// TIA Portal V19 export
DATA_BLOCK "AI SCALING DB"   // DB5
{ S7_Optimized_Access := 'TRUE' }
// stored: MemoryReserve 100
   VAR RETAIN
      MIN : Struct
         "SYRUP VESSEL TEMP SENSOR" : Real := -50.0;
         "PREMIXING VESSEL TEMP SENSOR" : Real := -50.0;
         "SUGAR VESSEL TEMP SENSOR" : Real := -50.0;
         "STEAM LINE_1 TEMP SENSOR" : Real := -50.0;
         "STEAM LINE_2 TEMP SENSOR" : Real := -50.0;
         "PRESSURE TRANSMITTER 1" : Real := -1.0;
         "PRESSURE TRANSMITTER 2" : Real := -1.0;
         "VACCIM TRANSMITTER 1" : Real := -750.0;
         "VACCIM TRANSMITTER 2" : Real := -750.0;
         "VACCUM TRANSMITTER 3" : Real := -750.0;
         "SYRUP LOAD CELL" : Real := 0.0;
         "PREMIXING LOAD CELL" : Real := 0.0;
         "SUGAR LOAD CELL" : Real := 0.0;
         "ULTRASONIC LEVEL SENSOR-1" : Real := 0.0;
         "ULTRASONIC LEVEL SENSOR-2" : Real := 0.0;
         "ULTRASONIC LEVEL SENSOR-3" : Real := 0.0;
      END_STRUCT;
      MAX : Struct
         "SYRUP VESSEL TEMP SENSOR" : Real := 250.0;
         "PREMIXING VESSEL TEMP SENSOR" : Real := 250.0;
         "SUGAR VESSEL TEMP SENSOR" : Real := 250.0;
         "STEAM LINE_1 TEMP SENSOR" : Real := 250.0;
         "STEAM LINE_2 TEMP SENSOR" : Real := 250.0;
         "PRESSURE TRANSMITTER 1" : Real := 5.0;
         "PRESSURE TRANSMITTER 2" : Real := 5.0;
         "VACCIM TRANSMITTER 1" : Real := 0.0;
         "VACCIM TRANSMITTER 2" : Real := 0.0;
         "VACCUM TRANSMITTER 3" : Real := 0.0;
         "SYRUP LOAD CELL" : Real := 5000.0;
         "PREMIXING LOAD CELL" : Real := 1500.0;
         "SUGAR LOAD CELL" : Real := 3750.0;
         "ULTRASONIC LEVEL SENSOR-1" : Real := 10000.0;
         "ULTRASONIC LEVEL SENSOR-2" : Real := 10000.0;
         "ULTRASONIC LEVEL SENSOR-3" : Real := 10000.0;
      END_STRUCT;
   END_VAR
   VAR
      PV : Struct
         "SYRUP VESSEL TEMP SENSOR" : Real;
         "PREMIXING VESSEL TEMP SENSOR" : Real;
         "SUGAR VESSEL TEMP SENSOR" : Real;
         "STEAM LINE_1 TEMP SENSOR" : Real;
         "STEAM LINE_2 TEMP SENSOR" : Real;
         "PRESSURE TRANSMITTER 1" : Real;
         "PRESSURE TRANSMITTER 2" : Real;
         "VACCIM TRANSMITTER 1" : Real;
         "VACCIM TRANSMITTER 2" : Real;
         "VACCUM TRANSMITTER 3" : Real;
         "SYRUP LOAD CELL" : Real;
         "PREMIXING LOAD CELL" : Real;
         "SUGAR LOAD CELL" : Real;
         "ULTRASONIC LEVEL SENSOR-1" : Real;
         "ULTRASONIC LEVEL SENSOR-2" : Real;
         "ULTRASONIC LEVEL SENSOR-3" : Real;
      END_STRUCT;
   END_VAR
BEGIN
END_DATA_BLOCK
